FUNCTION_BLOCK Demux (* Basic Function Block Type *)
  (* Standard: 61499-2 *)
  (* Version 0.0, 6/8/2016, Andrei, nxtControl GmbH, Template *)
  PACKAGE Main;
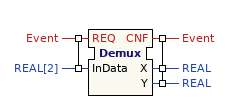
  EVENT_INPUT
    REQ WITH InData; (* Normal Execution Request *)
  END_EVENT
  EVENT_OUTPUT
    CNF WITH X, Y; (* Execution Confirmation *)
  END_EVENT
  VAR_INPUT
    InData : ARRAY [0..1] OF REAL; (* Input event qualifier *)
  END_VAR
  VAR_OUTPUT
    X : REAL; (* Output event qualifier *)
    Y : REAL;
  END_VAR
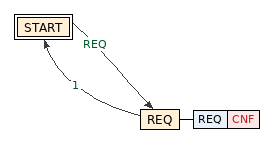
  EC_STATES
    START; (* Initial State *)
    REQ : REQ -> CNF; (* Normal execution *)
  END_STATES
  EC_TRANSITIONS
    START TO REQ := REQ;
    REQ TO START := 1;
  END_TRANSITIONS
  ALGORITHM REQ IN ST: (* Normally executed algorithm *)
X := InData[0];
Y := InData[1];
  END_ALGORITHM
END_FUNCTION_BLOCK
